INTERFACE IAbortableAction EXTENDS IAction

{attribute 'monitoring' := 'call'}
{attribute 'OPC.UA.DA.Property' := '1'}
{attribute 'OPC.UA.DA.Access' := '1'}
PROPERTY Aborted : BOOL
GET
END_GET
END_PROPERTY

{attribute 'monitoring' := 'call'}
{attribute 'OPC.UA.DA.Property' := '1'}
{attribute 'OPC.UA.DA.Access' := '1'}
PROPERTY Aborting : BOOL
GET
END_GET
END_PROPERTY

{attribute 'monitoring' := 'call'}
{attribute 'OPC.UA.DA.Property' := '1'}
{attribute 'OPC.UA.DA.Access' := '1'}
PROPERTY AbortReason : REFERENCE TO ERROR_MESSAGE
GET
END_GET
END_PROPERTY

METHOD RequestAbort
VAR_INPUT 
	reason : ERROR_MESSAGE;
END_VAR
END_METHOD

END_INTERFACE

(* stored: Version 1.1.0.1
   Itf IAbortableAction: Id {b0f9c97b-b928-4413-8759-73a11fb21302}
   Property Aborted: Id {6ef6c353-931c-4e44-9bed-97312556562d}
   Get Get: Id {70255aa6-718a-4eec-ae2a-07140208076f}
   Property Aborting: Id {fa6aaed9-b143-458f-9f53-372b8d41a320}
   Get Get: Id {68f85123-7faf-44dd-8da4-f3001d3270f1}
   Property AbortReason: Id {bb9081e9-96cd-46ff-932c-a25b56d0d11b}
   Get Get: Id {06007672-f17c-40c7-876c-d4f89dab3748}
   Method RequestAbort: Id {a65df189-274a-41f8-a347-a44b313e8bc2} *)
